FUNCTION_BLOCK FB_Robotersteuerung
VAR_INPUT
	rXpos : REAL;
	rYpos : REAL;
	rZpos : REAL;
	bGclose : BOOL;
END_VAR
VAR_OUTPUT
	eState : eBetriebszustand;
END_VAR
VAR
	nState : INT := 0;

	fbRoboterAchseX : FB_Roboterachsensteuerung;
	fbRoboterAchseY : FB_Roboterachsensteuerung;
	fbRoboterAchseZ : FB_Roboterachsensteuerung;
	fbRoboterAchseG : FB_Roboterachsensteuerung;
	bExecuteX: BOOL;
END_VAR

fbRoboterAchseX(
	bEnable:= bEnable, 
	bExecute:= , 
	rPosition:= , 
	bRefSens:= IFC_HW.bManEndXmin, 
	eState=> , 
	ax:= IFC_HW.ax_ManX);

fbRoboterAchseY(
	bEnable:= bEnable, 
	bExecute:= , 
	rPosition:= , 
	bRefSens:= IFC_HW.bManEndYmin, 
	eState=> , 
	ax:= IFC_HW.ax_ManY);
	
fbRoboterAchseZ(
	bEnable:= bEnable, 
	bExecute:= , 
	rPosition:= , 
	bRefSens:= IFC_HW.bManEndZmin, 
	eState=> , 
	ax:= IFC_HW.ax_ManZ);

fbRoboterAchseG(
	bEnable:= bEnable, 
	bExecute:= , 
	rPosition:= , 
	bRefSens:= IFC_HW.bManEndGmin, 
	eState=> , 
	ax:= IFC_HW.ax_ManG);
	
IF bExecuteX THEN
	METH_MoveXAxis(rXpos);
END_IF

	
CASE nState OF
	0: // OFF
	eState := eBetriebszustand.OFF;
	
	fbRoboterAchseX.bEnable := FALSE;
	fbRoboterAchseY.bEnable := FALSE;
	fbRoboterAchseZ.bEnable := FALSE;
	fbRoboterAchseG.bEnable := FALSE;
	
	IF bEnable THEN
		nState := 10;
	END_IF
	
	10: // INIT
	eState := eBetriebszustand.INIT;
	
	fbRoboterAchseX.bEnable := TRUE;
	fbRoboterAchseY.bEnable := TRUE;
	fbRoboterAchseZ.bEnable := TRUE;
	fbRoboterAchseG.bEnable := TRUE;
	
	IF (fbRoboterAchseX.eState = eBetriebszustand.READY) AND (fbRoboterAchseY.eState = eBetriebszustand.READY) AND 
	   (fbRoboterAchseZ.eState = eBetriebszustand.READY) AND (fbRoboterAchseG.eState = eBetriebszustand.READY) THEN   
	   nState := 20;
	END_IF
	
	20: // READY
	eState := eBetriebszustand.READY;
	
	IF bExecute THEN
		nState := 30;
	END_IF
	
	30: // PROD-ZAchse hoch
	eState := eBetriebszustand.PROD;
	fbRoboterAchseZ.rPosition := GVL_PosKinematic.pZoff;
	fbRoboterAchseZ.bExecute := TRUE;
	
	IF fbRoboterAchseZ.eState = eBetriebszustand.DONE THEN
		fbRoboterAchseZ.bExecute := FALSE;
		nstate := 31;
	END_IF
	
	31: // PROD-XYAchse bewegen
	eState := eBetriebszustand.PROD;
	
	fbRoboterAchseX.rPosition := rXpos;
	fbRoboterAchseY.rPosition := rYpos;
	fbRoboterAchseX.bExecute := TRUE;
	fbRoboterAchseY.bExecute := TRUE;
	
	IF (fbRoboterAchseZ.eState = eBetriebszustand.DONE) AND (fbRoboterAchseZ.eState = eBetriebszustand.DONE) THEN
		fbRoboterAchseX.bExecute := FALSE;
		fbRoboterAchseY.bExecute := FALSE;
		nstate := 32;
	END_IF
	
	32: // PROD-ZAchse bewegen
	eState := eBetriebszustand.PROD;
	IFC_HW.bManBrakeZ := TRUE;
	fbRoboterAchseZ.rPosition := rZpos;
	fbRoboterAchseZ.bExecute := TRUE;
	
	IF fbRoboterAchseZ.eState = eBetriebszustand.DONE THEN
		IFC_HW.bManBrakeZ := FALSE;
		fbRoboterAchseZ.bExecute := FALSE;
		nstate := 33;
	END_IF
	
	33: // PROD-GAchse bewegen
	eState := eBetriebszustand.PROD;
	IF bGclose THEN
		fbRoboterAchseG.rPosition := 0;
		fbRoboterAchseG.bExecute := TRUE;
		IFC_HW.bGripperClosed := TRUE;
	ELSE
		fbRoboterAchseG.rPosition := 0;
		fbRoboterAchseG.bExecute := TRUE;
		IFC_HW.bGripperClosed := FALSE;
	END_IF
		
	IF fbRoboterAchseG.eState = eBetriebszustand.DONE THEN
		fbRoboterAchseG.bExecute := FALSE;
		nstate := 33;
	END_IF
END_CASE

METHOD METH_MoveXAxis : BOOL
VAR_INPUT
	rPos	: REAL;
END_VAR
fbRoboterAchseX(
	bEnable:= bEnable, 
	bExecute:= TRUE, 
	rPosition:= rPos, 
	bRefSens:= IFC_HW.bManEndXmin, 
	eState=> , 
	ax:= IFC_HW.ax_ManX);
END_METHOD

END_FUNCTION_BLOCK

(* stored: Version 1.1.0.1, ProductVersion 3.1.4024.15
   POU FB_Robotersteuerung: Id {2dde4477-e1e2-4351-aa2e-f07033cc3dda}, SpecialFunc None
   Method METH_MoveXAxis: Id {1f2eac2d-5fae-468a-b6f4-7144b3654d8b} *)
